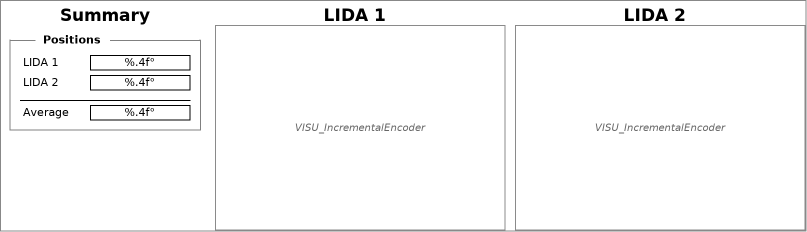
VISUALIZATION VISU_AxesElevationAxis_Lidas  // 807x232
VAR_IN_OUT
	ref : AxesElevationAxis;
    widget : AxesElevationAxisWidget;
END_VAR
    Label (215,0 280x30), "LIDA 1"
    Frame (215,25 290x205)
        shows VISU_IncrementalEncoder(ref := ref.parts.lida1, widget := widget.lida1)
    Label (515,0 280x30), "LIDA 2"
    Frame (515,25 290x205)
        shows VISU_IncrementalEncoder(ref := ref.parts.lida2, widget := widget.lida2)
    Label (10,0 190x30), "Summary"
    Label (40,30 65x20), "Positions"
    Polyline (110,40) (200,40) (200,130) (10,130) (10,40) (35,40)
    Label (20,55 90x15), "LIDA 1"
    Rectangle (90,55 100x15), "%.4f°", text variable: ref.lida1Position.degrees.value
    Rectangle (90,75 100x15), "%.4f°", text variable: ref.lida2Position.degrees.value
    Label (20,75 90x15), "LIDA 2"
    Label (20,105 90x15), "Average"
    Rectangle (90,105 100x15), "%.4f°", text variable: ref.lidaAveragePosition.degrees.value
    Line (20,100) (190,100)
END_VISUALIZATION

(* stored: Version 1.1.0.1, ProductVersion 3.1.4019.2
   Visu VISU_AxesElevationAxis_Lidas: Id {839a7743-20e0-4d3c-8876-10f9eb4cdb34} *)
